TYPE ST_RW :
STRUCT
	ReadFromNUC : BOOL:= FALSE;//enabling Read and Write can create unintended behaviour, consider feedback var
	WriteToNUC: BOOL:=FALSE ; //enabling Read and Write can create unintended behaviour, consider feedback var
END_STRUCT
END_TYPE

(* stored: Version 1.1.0.1, ProductVersion 3.1.4026.18
   DUT ST_RW: Id {edaf2162-0318-4345-beee-ca7bb42de741} *)
